FUNCTION_BLOCK WaterMonitor
  (* Standard: 61499-2 *)
  (* Version 0.2, 2003-12-05, JHC, Rockwell Automation, Renamed from NEWCOMPFB. *)
  (* Compiler header: package fb.rt.benchmarks.watermonitor; *)
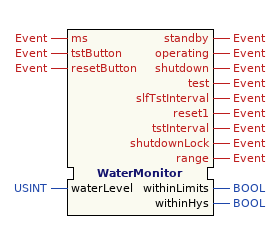
  EVENT_INPUT
    ms; (* millisecond *)
    tstButton;
    resetButton;
  END_EVENT
  EVENT_OUTPUT
    standby;
    operating;
    shutdown;
    test;
    slfTstInterval;
    reset1;
    tstInterval;
    shutdownLock;
    range;
  END_EVENT
  VAR_INPUT
    waterLevel : USINT;
  END_VAR
  VAR_OUTPUT
    withinLimits : BOOL;
    withinHys : BOOL;
  END_VAR
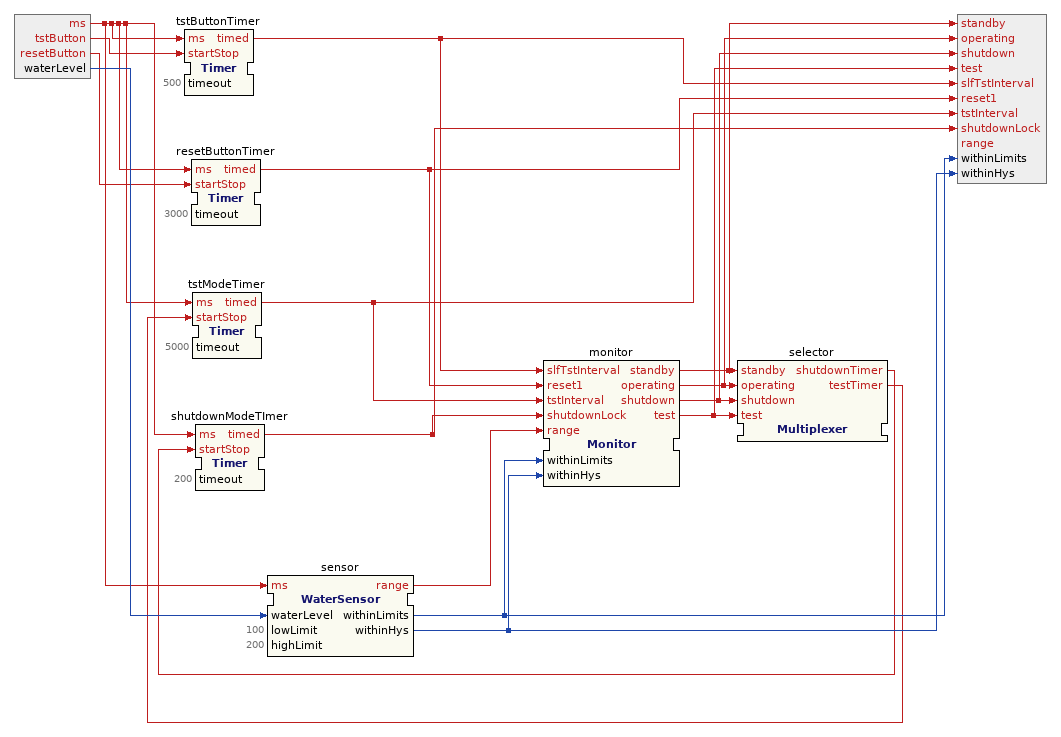
  FBS
    sensor : WaterSensor(lowLimit := 100, highLimit := 200);
    tstButtonTimer : Timer(timeout := 500);
    tstModeTimer : Timer(timeout := 5000);
    shutdownModeTImer : Timer(timeout := 200);
    resetButtonTimer : Timer(timeout := 3000);
    selector : Multiplexer;
    monitor : Monitor;
  END_FBS
  EVENT_CONNECTIONS
    ms TO sensor.ms;
    ms TO tstButtonTimer.ms;
    ms TO resetButtonTimer.ms;
    ms TO tstModeTimer.ms;
    tstButton TO tstButtonTimer.startStop;
    resetButton TO resetButtonTimer.startStop;
    tstButtonTimer.timed TO monitor.slfTstInterval;
    resetButtonTimer.timed TO monitor.reset1;
    tstModeTimer.timed TO monitor.tstInterval;
    shutdownModeTImer.timed TO monitor.shutdownLock;
    ms TO shutdownModeTImer.ms;
    sensor.range TO monitor.range;
    monitor.standby TO selector.standby;
    monitor.operating TO selector.operating;
    monitor.shutdown TO selector.shutdown;
    monitor.test TO selector.test;
    selector.shutdownTimer TO shutdownModeTImer.startStop;
    selector.testTimer TO tstModeTimer.startStop;
    monitor.standby TO standby;
    monitor.operating TO operating;
    monitor.shutdown TO shutdown;
    monitor.test TO test;
    tstButtonTimer.timed TO slfTstInterval;
    tstModeTimer.timed TO tstInterval;
    resetButtonTimer.timed TO reset1;
    shutdownModeTImer.timed TO shutdownLock;
  END_CONNECTIONS
  DATA_CONNECTIONS
    waterLevel TO sensor.waterLevel;
    sensor.withinLimits TO monitor.withinLimits;
    sensor.withinHys TO monitor.withinHys;
    sensor.withinLimits TO withinLimits;
    sensor.withinHys TO withinHys;
  END_CONNECTIONS
END_FUNCTION_BLOCK
